PROGRAM POU
VAR
	X1: BOOL;
	Y1: BOOL;
END_VAR

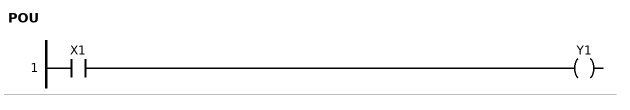
// NETWORK 1
Y1 := X1;

END_PROGRAM

(* stored: Version 1.1.0.1, ProductVersion 3.1.4024.11
   POU POU: Id {ae482b2a-8018-42d5-8ccd-8f2c44f52a8a}, SpecialFunc None *)
